{attribute 'qualified_only'}
{attribute 'strict'}
TYPE E_SourceType : 
(
	eLive := 0,
	eHistMQTT,
	eHistFile
) ;
END_TYPE

(* stored: DUT E_SourceType: Id 2e0b87a5-7110-44ef-83fa-7746ca338a73 *)
